Staubli VAL3: leftPos.pgx

public program leftPos(string x_sItem (dimensions=1), num x_nLength (dimensions=1), string& x_sResult[] (dimensions=1))
  local num i
  local num l_nLength
  local string l_sItem
begin
  //
  l_sItem=x_sItem
  //
  if len(l_sItem)!=getDisplayLen(l_sItem) and x_nLength>0
    for i=0 to len(x_sItem)-1
      l_nLength=l_nLength+getDisplayLen(left(l_sItem,1))
      l_sItem=right(l_sItem,len(l_sItem)-1)
      if l_nLength==x_nLength
        x_sResult=left(x_sItem,i+1)
        return
      else
        if l_nLength>x_nLength
          x_sResult=left(x_sItem,i)
          return
        endIf
      endIf
    endFor
    // else
  endIf
  x_sResult=left(x_sItem,max(x_nLength,0))
  // endIf
end
